VAR_GLOBAL CONSTANT
	///ctrl commands definitions
	///specific commands >200 - every command has to be a even number
	cCMD_RIGHT				: INT := 202;
	cCMD_LEFT				: INT := 204;
	
	///ctrl specific states definitions
	cSTA_SETOPERATIONMODE	: INT := 201;
	cSTA_RESETMOTORERROR	: INT := 203;
END_VAR

(* stored: Version 1.1.0.1, ProductVersion 3.1.0.19
   GVL UMC_CmdState: Id {fade76cb-e304-4f40-961e-87ad53eac9b3} *)
